FUNCTION_BLOCK T_ComponentsBlockHmiBlocked EXTENDS T_UnitTestBase
VAR
  list : T_ComponentsCollection;
  newComponent, newComponent2 : T_ComponentMock; 
  actual1, actual2 : BOOL;
END_VAR

// Arrange
list.AddComponent(newComponent);
list.AddComponent(newComponent2);

//Act
list.BlockHMIControl();

//Assert
actual1 := newComponent._hmiBlocked;
actual2 := newComponent2._hmiBlocked;

assertion.AssertEquals_BOOL(TRUE, actual1, 'actual1 := newComponent._hmiBlocked;');
assertion.AssertEquals_BOOL(TRUE, actual1, 'actual2 := newComponent2._hmiBlocked;');
TestFinished();

END_FUNCTION_BLOCK

(* stored: Version 1.1.0.1, ProductVersion 3.1.4024.12
   POU T_ComponentsBlockHmiBlocked: Id {b83b4f48-2528-42f3-b8f8-21dd09f25019}, SpecialFunc None *)
